(* IEC 61131-3 sources: Industry-PLC-LLM/data/PLCBEAD_repo/PLCBEAD_PLCEmbed-main/PLC-BEAD/Source/GEB/GEN_PULSE, 1 file *)

(* ---- GEN_PULSE.ST ---- *)
FUNCTION UDINT_TO_TIME2:TIME

	VAR_INPUT
		IN :	UDINT;
	END_VAR

	UDINT_TO_TIME2 := DINT_TO_TIME(UDINT_TO_DINT(IN));

END_FUNCTION

FUNCTION_BLOCK T_PLC_MS_block
	VAR_OUTPUT
		T_PLC_MS :	UDINT;
	END_VAR

	VAR
		PLC_TICKS_PER_SEC :	INT;
		PLC_SYS_TICK_CNT :	DINT;
	END_VAR

	VAR
		debug :	BOOL;(*Debug-Mode ON / OFF*)
		N :	INT;(*Debug-Faktor*)
		Offset :	UDINT;(*Debug-Offset*)
		temp :	DWORD := DWORD#1;(*Debug-Offset*)
		MODE :	BOOL;(*modus*)
		faktor :	UDINT;(*Systemtakt-Faktor*)
		init :	BOOL;
		v_plc_ticks_per_sec :	UDINT;
		base :	UDINT := UDINT#1000;
	END_VAR

	IF init = FALSE THEN
		v_plc_ticks_per_sec := INT_TO_UDINT(PLC_TICKS_PER_SEC);
		IF v_plc_ticks_per_sec = UDINT#1024 THEN
			faktor := UDINT#1;
			MODE := FALSE;
		ELSIF v_plc_ticks_per_sec > UDINT#0 THEN
			IF v_plc_ticks_per_sec <= base THEN
				faktor := base / v_plc_ticks_per_sec;
				MODE := FALSE;
			ELSE
				faktor := v_plc_ticks_per_sec / base;
				MODE := TRUE;
			END_IF;
		ELSE
			faktor := UDINT#1;
		END_IF;
		init := TRUE;
	END_IF;

	IF MODE THEN
		T_PLC_MS := DINT_TO_UDINT(PLC_SYS_TICK_CNT) / faktor;
	ELSE
		T_PLC_MS := DINT_TO_UDINT(PLC_SYS_TICK_CNT) * faktor;
	END_IF;

	IF debug THEN
		T_PLC_MS := (DWORD_TO_UDINT(SHL(UDINT_TO_DWORD(T_PLC_MS),N) OR SHL(temp,N)) - UDINT#1) + Offset;
	END_IF;

END_FUNCTION_BLOCK

FUNCTION_BLOCK GEN_PULSE_Block

	VAR_INPUT
		ENQ :	BOOL := TRUE;
		PTH :	TIME;
		PTL :	TIME;
	END_VAR

	VAR_OUTPUT
		Q :	BOOL;
	END_VAR

	VAR
		T_PLC_MS :	T_PLC_MS_block;
		TX :	TIME;
		tn :	TIME;
		init :	BOOL;
	END_VAR

	IF ENQ THEN
		T_PLC_MS();
		TX:= UDINT_TO_TIME(T_PLC_MS.T_PLC_MS);
		IF NOT init THEN init := TRUE; tn := TX; END_IF;
		IF SUB_TIME(TX, tn) >= SEL(Q, PTL, PTH) THEN
			tn := ADD_TIME(tn , SEL(Q, PTL, PTH));
			Q := NOT Q;
		END_IF;
	ELSE
		Q := FALSE;
		init := FALSE;
	END_IF;

END_FUNCTION_BLOCK

PROGRAM program0
  VAR
	ENQ :	BOOL := TRUE;
	PTH :	TIME;
	PTL :	TIME;
	Q :	BOOL;
	func_block : GEN_PULSE_Block;
  END_VAR
	func_block.ENQ  :=ENQ;
	func_block.PTH  :=PTH;
	func_block.PTL  :=PTL;
	func_block();
	Q := func_block.Q;

END_PROGRAM
